// SIMATIC S7-200 project (STEP 7-Micro/WIN), CPU 222 REL 01.22

ORGANIZATION_BLOCK PRINCIPAL:OB1
TITLE=COMENTARIOS DEL PROGRAMA
BEGIN
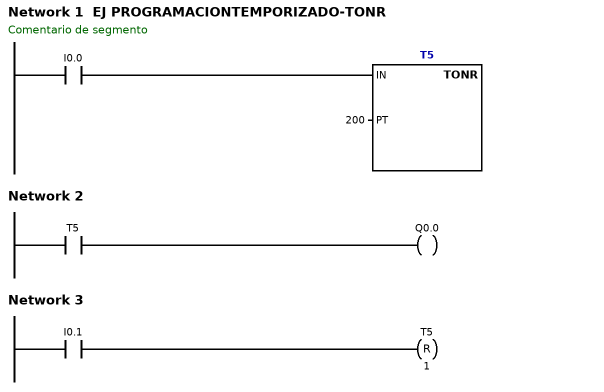
Network 1 // EJ PROGRAMACIONTEMPORIZADO-TONR

// Comentario de segmento
// (network saved uncompiled; LAD cells follow)
// row 0: c0 -| |- I0.0  c1 --  c2 --  c3 [TONR T5 IN:=power@row0, PT:=200]
// row 1: c3 [box]
Network 2
// (network saved uncompiled; LAD cells follow)
// row 0: c0 -| |- T5  c1 --  c2 --  c3 -( ) Q0.0
Network 3
// (network saved uncompiled; LAD cells follow)
// row 0: c0 -| |- I0.1  c1 --  c2 --  c3 -(R) T5, 1
END_ORGANIZATION_BLOCK
